// SIMATIC S7-200 SMART project (STEP 7-Micro/WIN SMART), CPU SR40

ORGANIZATION_BLOCK MAIN:OB1
TITLE=程序注释
BEGIN
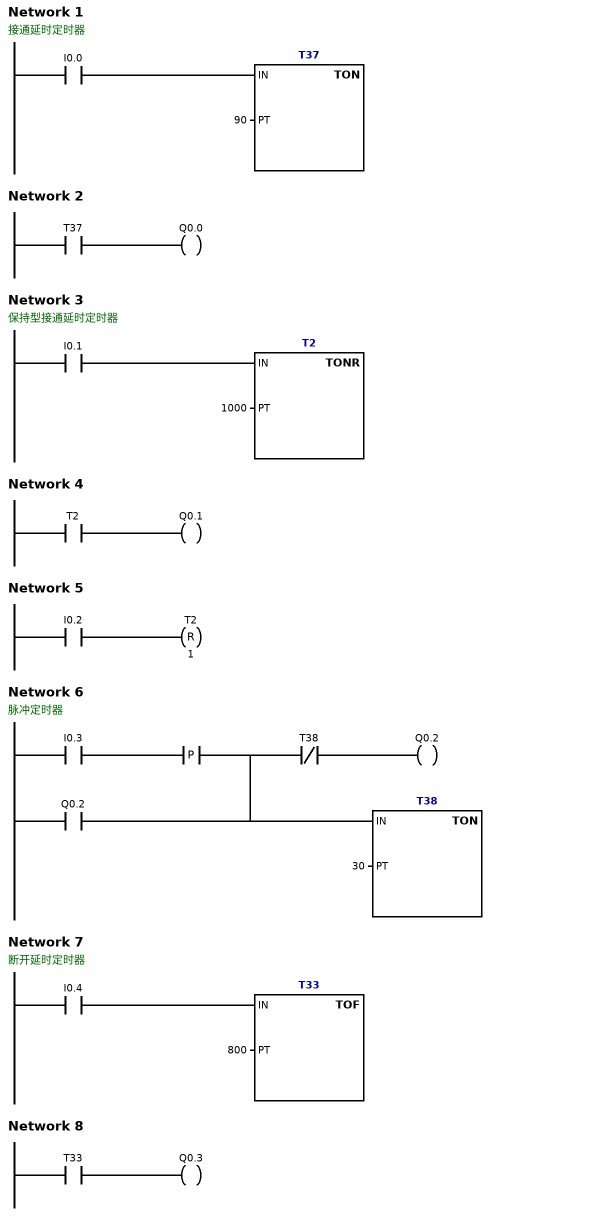
Network 1
// 接通延时定时器
LD     I0.0
TON    T37, 90
Network 2
LD     T37
=      Q0.0
Network 3
// 保持型接通延时定时器
LD     I0.1
TONR   T2, 1000
Network 4
LD     T2
=      Q0.1
Network 5
LD     I0.2
R      T2, 1
Network 6
// 脉冲定时器
LD     I0.3
EU
O      Q0.2
LPS
AN     T38
=      Q0.2
LPP
TON    T38, 30
Network 7
// 断开延时定时器
LD     I0.4
TOF    T33, 800
Network 8
LD     T33
=      Q0.3
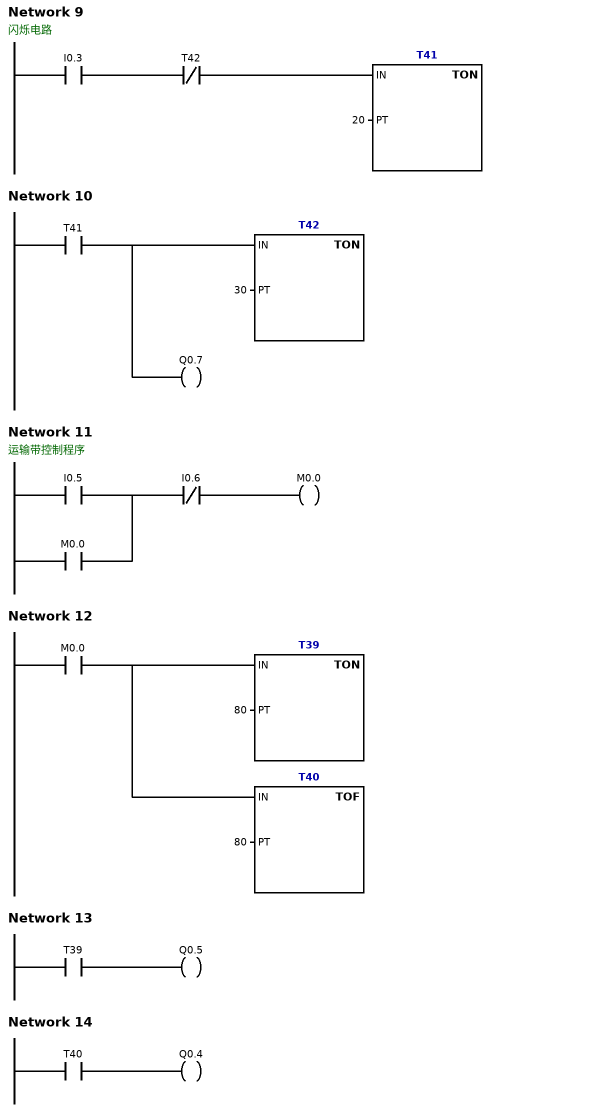
Network 9
// 闪烁电路
LD     I0.3
AN     T42
TON    T41, 20
Network 10
LD     T41
TON    T42, 30
=      Q0.7
Network 11
// 运输带控制程序
LD     I0.5
O      M0.0
AN     I0.6
=      M0.0
Network 12
LD     M0.0
TON    T39, 80
TOF    T40, 80
Network 13
LD     T39
=      Q0.5
Network 14
LD     T40
=      Q0.4
END_ORGANIZATION_BLOCK
